// TIA Portal V17 export
// export: Created 2025-06-26T06:33:58.9296998Z, ExportSetting WithDefaults, DisplayName Totally Integrated Automation Portal, DisplayVersion V17 Update 8, DisplayName TIA Portal Openness, DisplayVersion V17 Update 8, DisplayName TIA Portal Version Control Interface, DisplayVersion V17, DisplayName STEP 7 Professional, DisplayVersion V17 Update 8, DisplayName STEP 7 Safety, DisplayVersion V17 Update 6, DisplayName WinCC Advanced, DisplayVersion V17 Update 8
DATA_BLOCK "DB_CurrentSetting"   // DB21
{ S7_Optimized_Access := 'TRUE' }
AUTHOR : Heaten
VERSION : 0.1
// stored: AutoNumber false, DBAccessibleFromOPCUA true, IsOnlyStoredInLoadMemory false, IsRetainMemResEnabled false, IsWriteProtectedInAS false, MemoryReserve 0
   VAR RETAIN
      HeatSourceFlowLimit : Real := 0.0;   // [L/s] Heat source minimum volume flow
      HeatSinkFlowLimit : Real := 0.0;   // [L/s] Heat sink minimum volume flow
      "CAN-ModuleActive" : Bool := TRUE;   // 1 = do CAN comm, 0 = skip it
   END_VAR
BEGIN
END_DATA_BLOCK
